{attribute 'TcGenerated'}
// This function has been automatically generated from the project information.
VAR_GLOBAL CONSTANT
	{attribute 'const_non_replaced'}
	{attribute 'linkalways'}
	stLibVersion_PMPS : ST_LibVersion := (iMajor := 0, iMinor := 0, iBuild := 0, iRevision := 0, sVersion := '0.0.0');
END_VAR

(* stored: Version 1.1.0.1, ProductVersion 3.1.4022.12
   GVL Global_Version: Id {e5d19ae2-5eaa-0d66-1d74-00b138db6472} *)
